(* Logix 5000 project; controller KTC_LAB4_PT2 vendor 1 type 14 code 150 rev 30.11; software revision 30.00 *)

TASK MainTask (continuous, watchdog 500 ms) : MainProgram

MODULES
   Local : vendor 1 type 14 code 150 (Compact 0, rev 30.11)
      Counters : Embedded (Compact 3, rev 1.1, Output RPI 20 ms)
      Discrete_IO : Embedded (Compact 1, rev 3.1, Output RPI 20 ms)
      Analog_IO : Embedded (Compact 2, rev 1.1, Output RPI 80 ms)
END_MODULES

PROGRAM MainProgram   (* main routine MainRoutine *)
VAR
   PL0 : ALIAS FOR Local:1:O.Data.0;   // LIGHT 0 PART A
   PL1 : ALIAS FOR Local:1:O.Data.1;   // LIGHT 1 PART B
   PL2 : ALIAS FOR Local:1:O.Data.2;   // LIGHT 2 PART C
   PL3 : ALIAS FOR Local:1:O.Data.3;   // LIGHT 3 PART E
   PL4 : ALIAS FOR Local:1:O.Data.4;   // LIGHT 4 PROB 3
   SW4 : ALIAS FOR Local:1:I.Data.4;   // A
   SW5 : ALIAS FOR Local:1:I.Data.5;   // B
   SW6 : ALIAS FOR Local:1:I.Data.6;   // C
   SW7 : ALIAS FOR Local:1:I.Data.7;   // D
END_VAR

ROUTINE MainRoutine   (* ladder *)
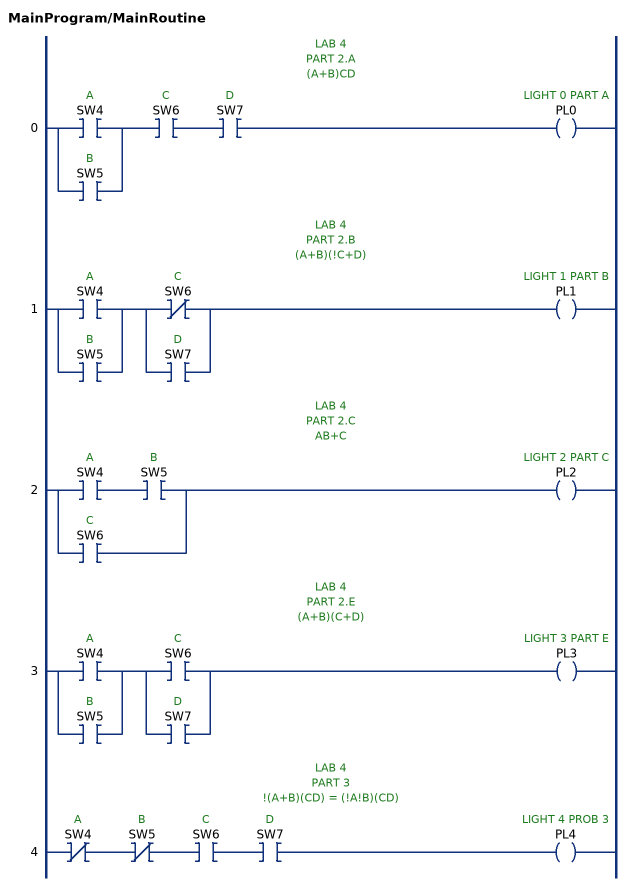
   // LAB 4
   // PART 2.A
   // (A+B)CD
   0: [XIC(SW4) ,XIC(SW5) ]XIC(SW6)XIC(SW7)OTE(PL0);
   // LAB 4
   // PART 2.B
   // (A+B)(!C+D)
   1: [XIC(SW4) ,XIC(SW5) ][XIO(SW6) ,XIC(SW7) ]OTE(PL1);
   // LAB 4
   // PART 2.C
   // AB+C
   2: [XIC(SW4) XIC(SW5) ,XIC(SW6) ]OTE(PL2);
   // LAB 4
   // PART 2.E
   // (A+B)(C+D)
   3: [XIC(SW4) ,XIC(SW5) ][XIC(SW6) ,XIC(SW7) ]OTE(PL3);
   // LAB 4
   // PART 3
   // !(A+B)(CD) = (!A!B)(CD)
   4: XIO(SW4)XIO(SW5)XIC(SW6)XIC(SW7)OTE(PL4);
END_ROUTINE
END_PROGRAM
